// TIA Portal V18 export
DATA_BLOCK "CappingStation_CounterON"   // DB61
{ S7_Optimized_Access := 'TRUE' }
// stored: AutoNumber true, DBAccessibleFromOPCUA true, InstanceOfName IEC_DCOUNTER, OfSystemLibElement IEC_DCOUNTER, OfSystemLibVersion 1.0
"IEC_DCOUNTER"
   // VAR RETAIN
   //    CU : Bool;
   //    CD : Bool;
   //    R : Bool;
   //    LD : Bool;
   //    QU : Bool;
   //    QD : Bool;
   //    PV : DInt;
   //    CV : DInt;
   // END_VAR
BEGIN
END_DATA_BLOCK
